{attribute 'no_explicit_call' := 'do not call this POU directly'} 
FUNCTION_BLOCK AnalogOutput IMPLEMENTS I_AnalogChannel
VAR_INPUT
END_VAR
VAR_OUTPUT
END_VAR
VAR
    {attribute 'TcInitSymbol'}
	ID:				STRING(25);
	Channel			AT%I*: INT;
END_VAR

METHOD FB_init : BOOL
VAR_INPUT
	bInitRetains : BOOL; // if TRUE, the retain variables are initialized (warm start / cold start)
	bInCopyCode : BOOL;  // if TRUE, the instance afterwards gets moved into the copy code (online change)
	ID:				STRING(25);
END_VAR
THIS^.ID:= ID;
END_METHOD

PROPERTY PUBLIC P_ID : String(25)
GET
P_ID:= ID;
END_GET
END_PROPERTY

PROPERTY P_State : EPlcMappingStatus
GET
P_State:= F_GetMappingStatus(ADR(Channel), SIZEOF(INT));
END_GET
END_PROPERTY

PROPERTY PUBLIC P_Value : Lreal
GET
P_Value:= INT_TO_LREAL(Channel);
END_GET
SET // PUBLIC
Channel:= LREAL_TO_INT(P_Value);
END_SET
END_PROPERTY

END_FUNCTION_BLOCK

(* stored: Version 1.1.0.1
   POU AnalogOutput: Id {7f986a17-ab6d-03bd-1c98-a964e10e1b1e}, SpecialFunc None
   Method FB_init: Id {fc427ba8-2be8-0fc8-1ba1-4c059d06ed11}
   Property P_ID: Id {030e0eaa-c0a4-09b4-3514-eb98d5fd7097}
   Get Get: Id {25c131a6-5f18-024c-3a39-ec1eed18a7fb}
   Property P_State: Id {8b895335-f806-0732-379a-cc62bed8728a}
   Get Get: Id {4dec217a-b567-08c7-1859-de70a267d3b2}
   Property P_Value: Id {a955e2d0-0b5a-083c-1316-087f566ed02a}
   Get Get: Id {07e3405e-d65d-019d-0fb5-767131610386}
   Set Set: Id {55ec4fbd-3d98-0de0-2d45-228ab7d2678e} *)
